# EPICS substitutions: indfurnSup/indfurn_thermocouple_faults.substitutions
file indfurn_pid.template {

pattern {PORT, P, ROOT, CMD}
{"\$(PORT)", "\$(P)", "\$(P)TC1FAULTS", "getTcFault"}
{"\$(PORT)", "\$(P)", "\$(P)TC2FAULTS", "getTc2Fault"}
}
